% RSLogix 500 project Multi-Position Valve Control System with Emergency Reset.RSS, saved by version 8.30.00.16 %
PROJECT "P4 "    % processor: Bul.1763 MicroLogix 1100 Series B %

PROGRAM FILES
  LAD 2   4 rungs
  LAD 3 "IO"  7 rungs
  LAD 4 "CTRL"  11 rungs
  LAD 5 "POSITION"  10 rungs

DATA FILES
  O0 OUTPUT  4 elements
  I1 INPUT  6 elements
  S2 STATUS  66 elements
  B3 BINARY  2 elements
  T4 TIMER  3 elements
  C5 COUNTER  1 elements
  R6 CONTROL  1 elements
  N7 INTEGER  2 elements
  F8 FLOAT  1 elements

LADDER 2
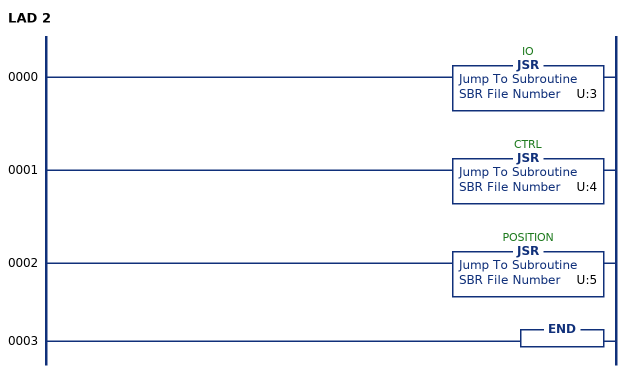
% Rung: 0 %
SOR JSR U:3 EOR
%   U:3  "IO" %
% Rung: 1 %
SOR JSR U:4 EOR
%   U:4  "CTRL" %
% Rung: 2 %
SOR JSR U:5 EOR
%   U:5  "POSITION" %
% Rung: 3 %
SOR END EOR

LADDER 3 "IO"
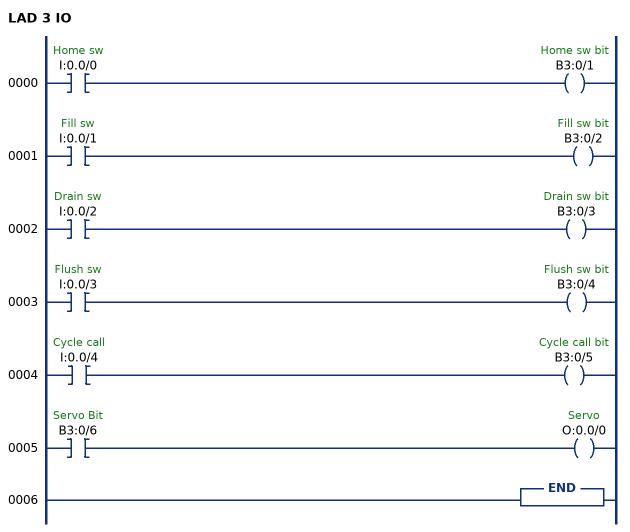
% Rung: 0 %
SOR XIC I:0.0/0 OTE B3:0/1 EOR
%   I:0.0/0  "Home sw" %
%   B3:0/1  "Home sw bit" %
% Rung: 1 %
SOR XIC I:0.0/1 OTE B3:0/2 EOR
%   I:0.0/1  "Fill sw" %
%   B3:0/2  "Fill sw bit" %
% Rung: 2 %
SOR XIC I:0.0/2 OTE B3:0/3 EOR
%   I:0.0/2  "Drain sw" %
%   B3:0/3  "Drain sw bit" %
% Rung: 3 %
SOR XIC I:0.0/3 OTE B3:0/4 EOR
%   I:0.0/3  "Flush sw" %
%   B3:0/4  "Flush sw bit" %
% Rung: 4 %
SOR XIC I:0.0/4 OTE B3:0/5 EOR
%   I:0.0/4  "Cycle call" %
%   B3:0/5  "Cycle call bit" %
% Rung: 5 %
SOR XIC B3:0/6 OTE O:0.0/0 EOR
%   B3:0/6  "Servo Bit" %
%   O:0.0/0  "Servo" %
% Rung: 6 %
SOR END EOR

LADDER 4 "CTRL"
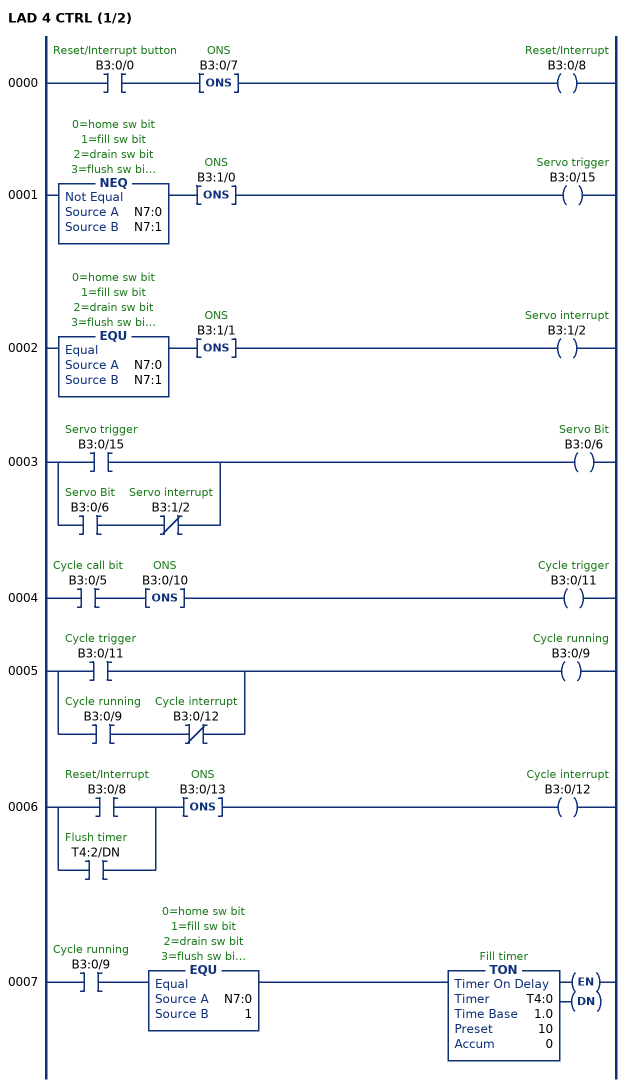
% Rung: 0 %
SOR XIC B3:0/0 ONS B3:0/7 OTE B3:0/8 EOR
%   B3:0/0  "Reset/Interrupt button" %
%   B3:0/7  "ONS" %
%   B3:0/8  "Reset/Interrupt" %
% Rung: 1 %
SOR NEQ N7:0 N7:1 ONS B3:1/0 OTE B3:0/15 EOR
%   N7:0  "0=home sw bit 1=fill sw bit 2=drain sw bit 3=flush sw bit 4=Travelling" %
%   N7:1  "Desired 0=home sw bit 1=fill sw bit 2=drain sw bit 3=flush sw bit" %
%   B3:1/0  "ONS" %
%   B3:0/15  "Servo trigger" %
% Rung: 2 %
SOR EQU N7:0 N7:1 ONS B3:1/1 OTE B3:1/2 EOR
%   N7:0  "0=home sw bit 1=fill sw bit 2=drain sw bit 3=flush sw bit 4=Travelling" %
%   N7:1  "Desired 0=home sw bit 1=fill sw bit 2=drain sw bit 3=flush sw bit" %
%   B3:1/1  "ONS" %
%   B3:1/2  "Servo interrupt" %
% Rung: 3 %
SOR BST XIC B3:0/15 NXB XIC B3:0/6 XIO B3:1/2 BND OTE B3:0/6 EOR
%   B3:0/15  "Servo trigger" %
%   B3:0/6  "Servo Bit" %
%   B3:1/2  "Servo interrupt" %
% Rung: 4 %
SOR XIC B3:0/5 ONS B3:0/10 OTE B3:0/11 EOR
%   B3:0/5  "Cycle call bit" %
%   B3:0/10  "ONS" %
%   B3:0/11  "Cycle trigger" %
% Rung: 5 %
SOR BST XIC B3:0/11 NXB XIC B3:0/9 XIO B3:0/12 BND OTE B3:0/9 EOR
%   B3:0/11  "Cycle trigger" %
%   B3:0/9  "Cycle running" %
%   B3:0/12  "Cycle interrupt" %
% Rung: 6 %
SOR BST XIC B3:0/8 NXB XIC T4:2/DN BND ONS B3:0/13 OTE B3:0/12 EOR
%   B3:0/8  "Reset/Interrupt" %
%   T4:2/DN  "Flush timer" %
%   B3:0/13  "ONS" %
%   B3:0/12  "Cycle interrupt" %
% Rung: 7 %
SOR XIC B3:0/9 EQU N7:0 1 TON T4:0 1.0 10 0 EOR
%   B3:0/9  "Cycle running" %
%   N7:0  "0=home sw bit 1=fill sw bit 2=drain sw bit 3=flush sw bit 4=Travelling" %
%   T4:0  "Fill timer" %

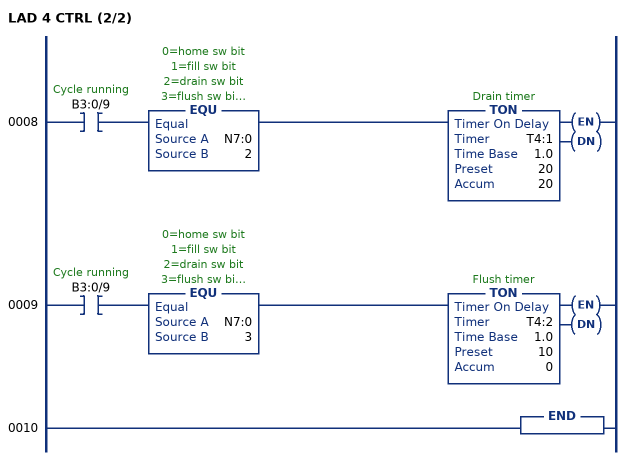
% Rung: 8 %
SOR XIC B3:0/9 EQU N7:0 2 TON T4:1 1.0 20 20 EOR
%   B3:0/9  "Cycle running" %
%   N7:0  "0=home sw bit 1=fill sw bit 2=drain sw bit 3=flush sw bit 4=Travelling" %
%   T4:1  "Drain timer" %
% Rung: 9 %
SOR XIC B3:0/9 EQU N7:0 3 TON T4:2 1.0 10 0 EOR
%   B3:0/9  "Cycle running" %
%   N7:0  "0=home sw bit 1=fill sw bit 2=drain sw bit 3=flush sw bit 4=Travelling" %
%   T4:2  "Flush timer" %
% Rung: 10 %
SOR END EOR

LADDER 5 "POSITION"
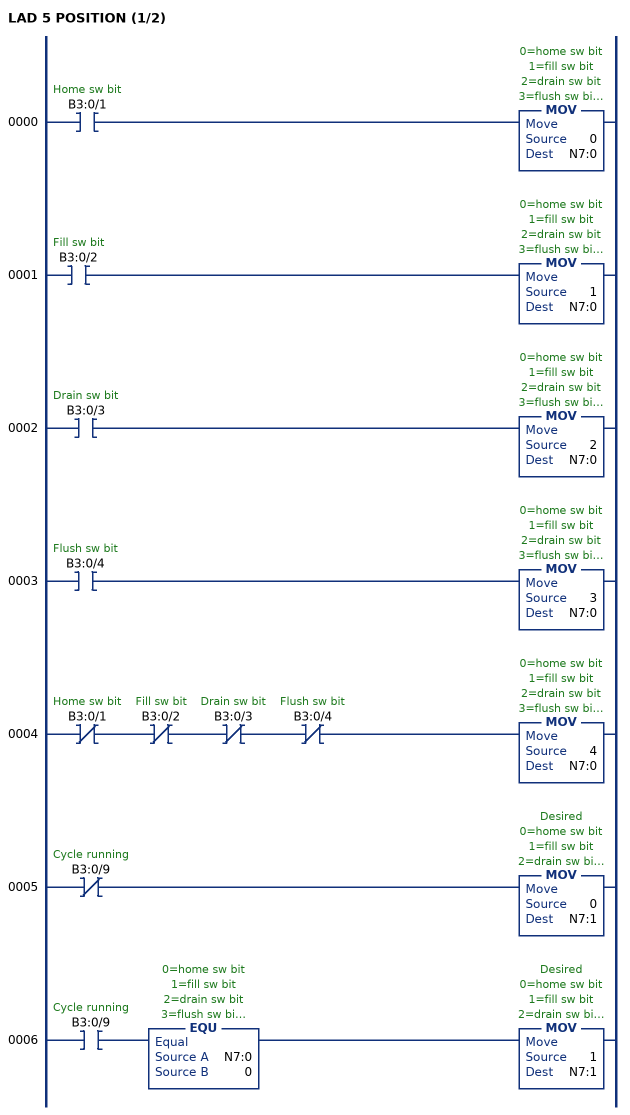
% Rung: 0 %
SOR XIC B3:0/1 MOV 0 N7:0 EOR
%   B3:0/1  "Home sw bit" %
%   N7:0  "0=home sw bit 1=fill sw bit 2=drain sw bit 3=flush sw bit 4=Travelling" %
% Rung: 1 %
SOR XIC B3:0/2 MOV 1 N7:0 EOR
%   B3:0/2  "Fill sw bit" %
%   N7:0  "0=home sw bit 1=fill sw bit 2=drain sw bit 3=flush sw bit 4=Travelling" %
% Rung: 2 %
SOR XIC B3:0/3 MOV 2 N7:0 EOR
%   B3:0/3  "Drain sw bit" %
%   N7:0  "0=home sw bit 1=fill sw bit 2=drain sw bit 3=flush sw bit 4=Travelling" %
% Rung: 3 %
SOR XIC B3:0/4 MOV 3 N7:0 EOR
%   B3:0/4  "Flush sw bit" %
%   N7:0  "0=home sw bit 1=fill sw bit 2=drain sw bit 3=flush sw bit 4=Travelling" %
% Rung: 4 %
SOR XIO B3:0/1 XIO B3:0/2 XIO B3:0/3 XIO B3:0/4 MOV 4 N7:0 EOR
%   B3:0/1  "Home sw bit" %
%   B3:0/2  "Fill sw bit" %
%   B3:0/3  "Drain sw bit" %
%   B3:0/4  "Flush sw bit" %
%   N7:0  "0=home sw bit 1=fill sw bit 2=drain sw bit 3=flush sw bit 4=Travelling" %
% Rung: 5 %
SOR XIO B3:0/9 MOV 0 N7:1 EOR
%   B3:0/9  "Cycle running" %
%   N7:1  "Desired 0=home sw bit 1=fill sw bit 2=drain sw bit 3=flush sw bit" %
% Rung: 6 %
SOR XIC B3:0/9 EQU N7:0 0 MOV 1 N7:1 EOR
%   B3:0/9  "Cycle running" %
%   N7:0  "0=home sw bit 1=fill sw bit 2=drain sw bit 3=flush sw bit 4=Travelling" %
%   N7:1  "Desired 0=home sw bit 1=fill sw bit 2=drain sw bit 3=flush sw bit" %

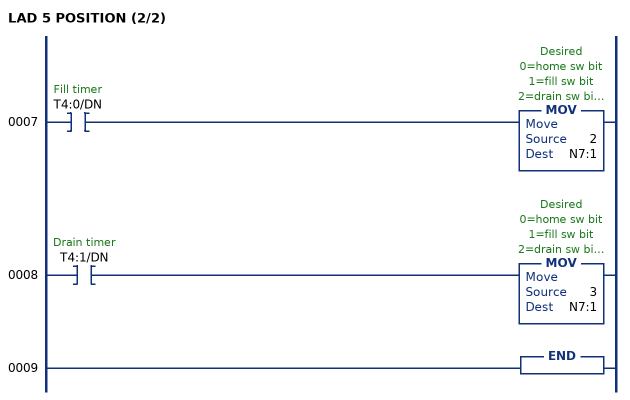
% Rung: 7 %
SOR XIC T4:0/DN MOV 2 N7:1 EOR
%   T4:0/DN  "Fill timer" %
%   N7:1  "Desired 0=home sw bit 1=fill sw bit 2=drain sw bit 3=flush sw bit" %
% Rung: 8 %
SOR XIC T4:1/DN MOV 3 N7:1 EOR
%   T4:1/DN  "Drain timer" %
%   N7:1  "Desired 0=home sw bit 1=fill sw bit 2=drain sw bit 3=flush sw bit" %
% Rung: 9 %
SOR END EOR

OTHER DOCUMENTED ADDRESSES
  B3:0/14  "Cycle Complete"

DATA TABLE (non-zero values as saved)
DATA B3
% B3:0 % 0X2240 0X0001
DATA T4
% .PRE .ACC %
% T4:0 % 10 0
% T4:1 % 20 20
% T4:2 % 10 0
